TYPE ST_SafetyDiagInfo :
STRUCT
	usintState			:USINT;
	usintDummy			:USINT;
	uintDiag			:UINT;
	usintDiag			:USINT;
END_STRUCT
END_TYPE

(* stored: Version 1.1.0.1, ProductVersion 3.1.4024.12
   DUT ST_SafetyDiagInfo: Id {f75173e3-a6d8-4adc-91d4-995439b5792a} *)
